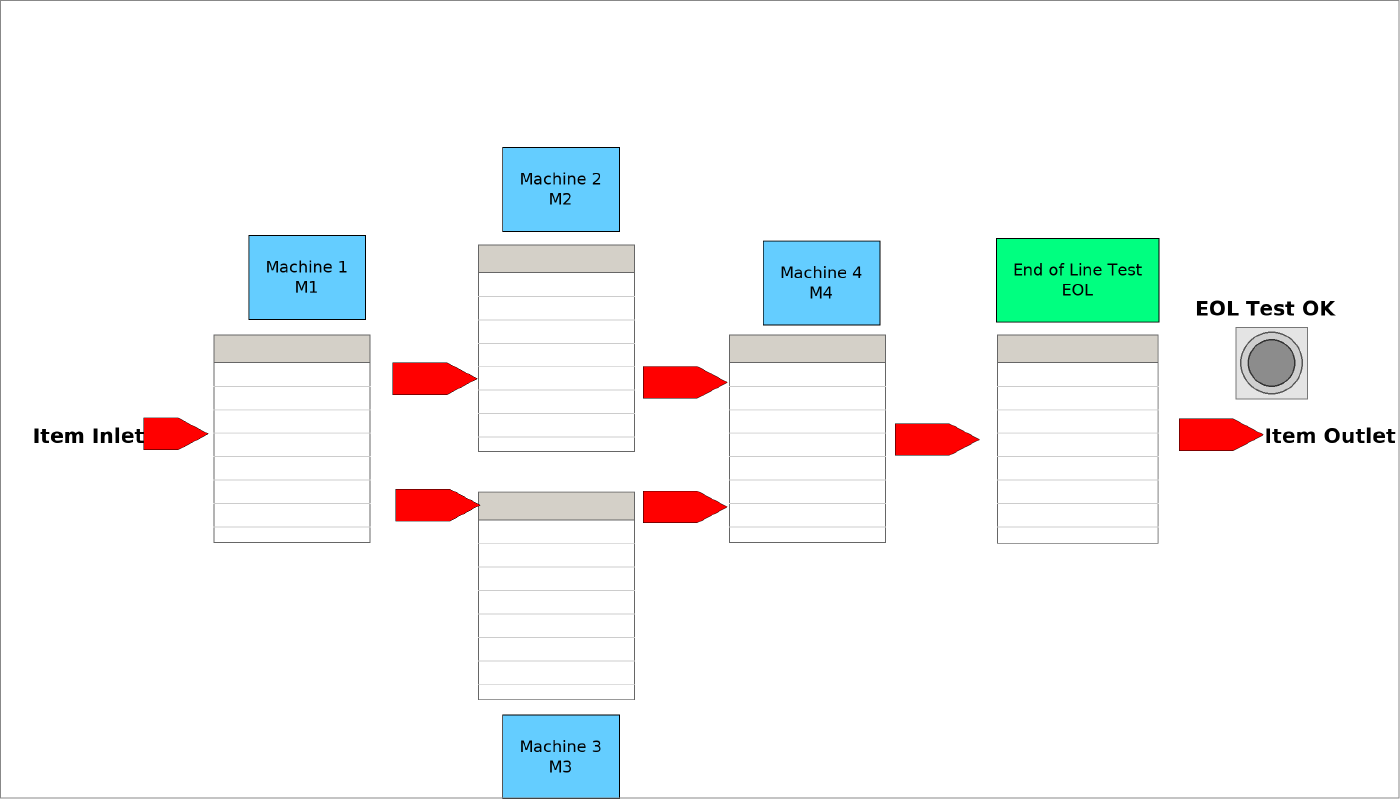
VISUALIZATION Visu1  // 1494x853
    Table (228,357 167x222), data array: MAIN.Fifo01.Queue
        p3854506369: MAIN.Fifo01.Queue[INDEX]
        p2232123230: FIFO_TEST.Fifo01.Queue[INDEX]
    Table (510,261 167x221), data array: MAIN.Fifo02.Queue
        p3854506369: MAIN.Fifo02.Queue[INDEX]
        p2232123230: FIFO_TEST.Fifo02.Queue[INDEX]
    Table (510,525 167x222), data array: MAIN.Fifo03.Queue
        p3854506369: MAIN.Fifo03.Queue[INDEX]
        p2232123230: FIFO_TEST.Fifo03.Queue[INDEX]
    Table (778,357 167x222), data array: MAIN.Fifo04.Queue
        p3854506369: MAIN.Fifo04.Queue[INDEX]
        p2232123230: FIFO_TEST.Fifo04.Queue[INDEX]
    Table (1064,357 172x223), data array: MAIN.FifoEol.Queue
        p3854506369: MAIN.FifoEol.Queue[INDEX]
        p2232123230: FIFO_TEST.Fifo05.Queue[INDEX]
    PushSwitch (1315,349 84x77), variable: MAIN.Eol, behaviour: TAP, style: Switch-PushSwitch-Gray
    Polygon (153,446) (153,480) (190,480) (222,463) (190,446), invisible if: NOT MAIN.tpIn.Q
    Polygon (419,387) (419,421) (477,421) (509,404) (477,387), invisible if: NOT MAIN.tpM02In.Q
    Polygon (422,522) (422,556) (480,556) (512,539) (480,522), invisible if: NOT MAIN.tpM03In.Q
    Polygon (686,391) (686,425) (744,425) (776,408) (744,391), invisible if: NOT MAIN.tpM02Out.Q
    Polygon (686,524) (686,558) (744,558) (776,541) (744,524), invisible if: NOT MAIN.tpM03Out.Q
    Polygon (955,452) (955,486) (1013,486) (1045,469) (1013,452), invisible if: NOT MAIN.tpM04Out.Q
    Polygon (1258,447) (1258,481) (1316,481) (1348,464) (1316,447), invisible if: NOT MAIN.tpEolOut.Q
    RoundedRectangle (265,251 125x90), "Machine 1 M1"
    RoundedRectangle (536,157 125x90), "Machine 2 M2"
    RoundedRectangle (536,763 125x90), "Machine 3 M3"
    RoundedRectangle (814,257 125x90), "Machine 4 M4"
    RoundedRectangle (1063,254 174x90), "End of Line Test EOL"
    Label (1264,308 172x43), "EOL Test OK"
    Label (20,444 149x43), "Item Inlet"
    Label (1345,444 149x43), "Item Outlet"
END_VISUALIZATION

(* stored: Version 1.1.0.1, ProductVersion 3.1.4024.15
   Visu Visu1: Id {f3733907-e397-48b9-b1d2-7db9de8c8173} *)
